(* IEC 61131-3 sources: AxTestProject/Program/LStandardLibrary/Math, 2 files *)

(* ---- Defaults.st ---- *)
NAMESPACE System.Math

    NAMESPACE Const

        FUNCTION PI : LReal
                PI := 3.1415926535897932384626433832795;
        END_FUNCTION

        FUNCTION MaxInt : INT
                MaxInt := 32767;
        END_FUNCTION

        FUNCTION MinInt : INT
                MinInt := -32768;
        END_FUNCTION

        FUNCTION MaxDInt : DINT
                MaxDInt := DINT#2147483647;
        END_FUNCTION

        FUNCTION MinDInt : DINT
                MinDInt := DINT#-2147483647;
        END_FUNCTION

    END_NAMESPACE

END_NAMESPACE

(* ---- DefaultsTest.st ---- *)
NAMESPACE System.Math.Test

    {Test}
    FUNCTION Constants
        VAR_INPUT
        END_VAR
        VAR_TEMP
        END_VAR

        Assert_Equal_LREAL(expected := 3.1415926535897932384626433832795, actual := System.Math.Const.PI());
        Assert_Equal_INT(expected := 32767, actual := System.Math.Const.MaxInt());
        Assert_Equal_INT(expected := -32768, actual := System.Math.Const.MinInt());

        Assert_Equal_DINT(expected := DINT#2147483647, actual := System.Math.Const.MaxDInt());
        Assert_Equal_DINT(expected := DINT#-2147483647, actual := System.Math.Const.MinDInt());

    END_FUNCTION

END_NAMESPACE
